{attribute 'pack_mode' := '1'}
TYPE ST_StatusPath :
STRUCT
	nPathID						: UINT;
	sCellID						: STRING(30);
	bPathPresent				: BOOL;
	nState						: UINT;			// E_MMPathState
	nMotionStatus				: UINT;			// E_MMPathMotionStatus
END_STRUCT
END_TYPE

(* stored: Version 1.1.0.1, ProductVersion 3.1.4024.5
   DUT ST_StatusPath: Id {5a374d6c-d992-4064-96aa-29e8c17b68cd} *)
